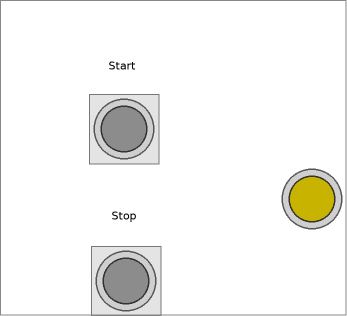
VISUALIZATION Visualization  // 347x316
    Lamp1 (277,164 70x70), variable: MAIN.Motor, style: Lamp-Lamp1-Yellow
    PushSwitch (89,94 70x70), variable: MAIN.PBSTart, behaviour: TAP, style: Switch-PushSwitch-Gray
    PushSwitch (91,246 70x70), variable: MAIN.PBStop, behaviour: TAP, style: Switch-PushSwitch-Gray
    Label (47,51 150x30), "Start"
    Label (49,201 150x30), "Stop"
END_VISUALIZATION

(* stored: Version 1.1.0.1, ProductVersion 3.1.4024.12
   Visu Visualization: Id {d9f1f7b6-f8b4-498c-8fe9-cf22e06fb6b8} *)
